PROGRAM Stn3
VAR

	start3: BOOL;
	reset3: BOOL;

	Stn3ProcessFE: F_TRIG;
	Stn3ProcessRE: R_TRIG;
	bCutStn3ProcessHalt: BOOL;
	DoorClose3: R_TRIG;
	bStn3DoorClamp: BOOL;
END_VAR
VAR // added by the converter: edge detectors and wires of the graphical bodies
    _w1, _w2 : ANY;
    _w3 : BOOL;
END_VAR

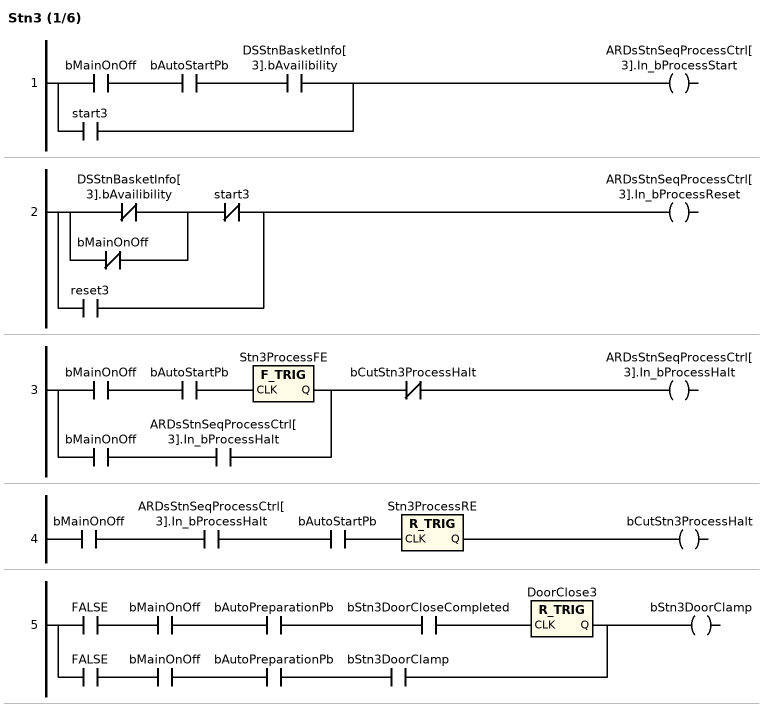
// NETWORK 1
ARDsStnSeqProcessCtrl[3].In_bProcessStart := bMainOnOff AND bAutoStartPb AND DSStnBasketInfo[3].bAvailibility OR start3;

// NETWORK 2
ARDsStnSeqProcessCtrl[3].In_bProcessReset := (NOT DSStnBasketInfo[3].bAvailibility OR NOT bMainOnOff) AND NOT start3 OR reset3;

// NETWORK 3
Stn3ProcessFE(CLK := bMainOnOff AND bAutoStartPb); // F_TRIG
ARDsStnSeqProcessCtrl[3].In_bProcessHalt := (Stn3ProcessFE.Q OR bMainOnOff AND ARDsStnSeqProcessCtrl[3].In_bProcessHalt) AND NOT bCutStn3ProcessHalt;

// NETWORK 4
Stn3ProcessRE(CLK := bMainOnOff AND ARDsStnSeqProcessCtrl[3].In_bProcessHalt AND bAutoStartPb); // R_TRIG
bCutStn3ProcessHalt := Stn3ProcessRE.Q;

// NETWORK 5
DoorClose3(CLK := (FALSE AND bMainOnOff AND bAutoPreparationPb) AND bStn3DoorCloseCompleted); // R_TRIG
bStn3DoorClamp := DoorClose3.Q OR (FALSE AND bMainOnOff AND bAutoPreparationPb) AND bStn3DoorClamp;

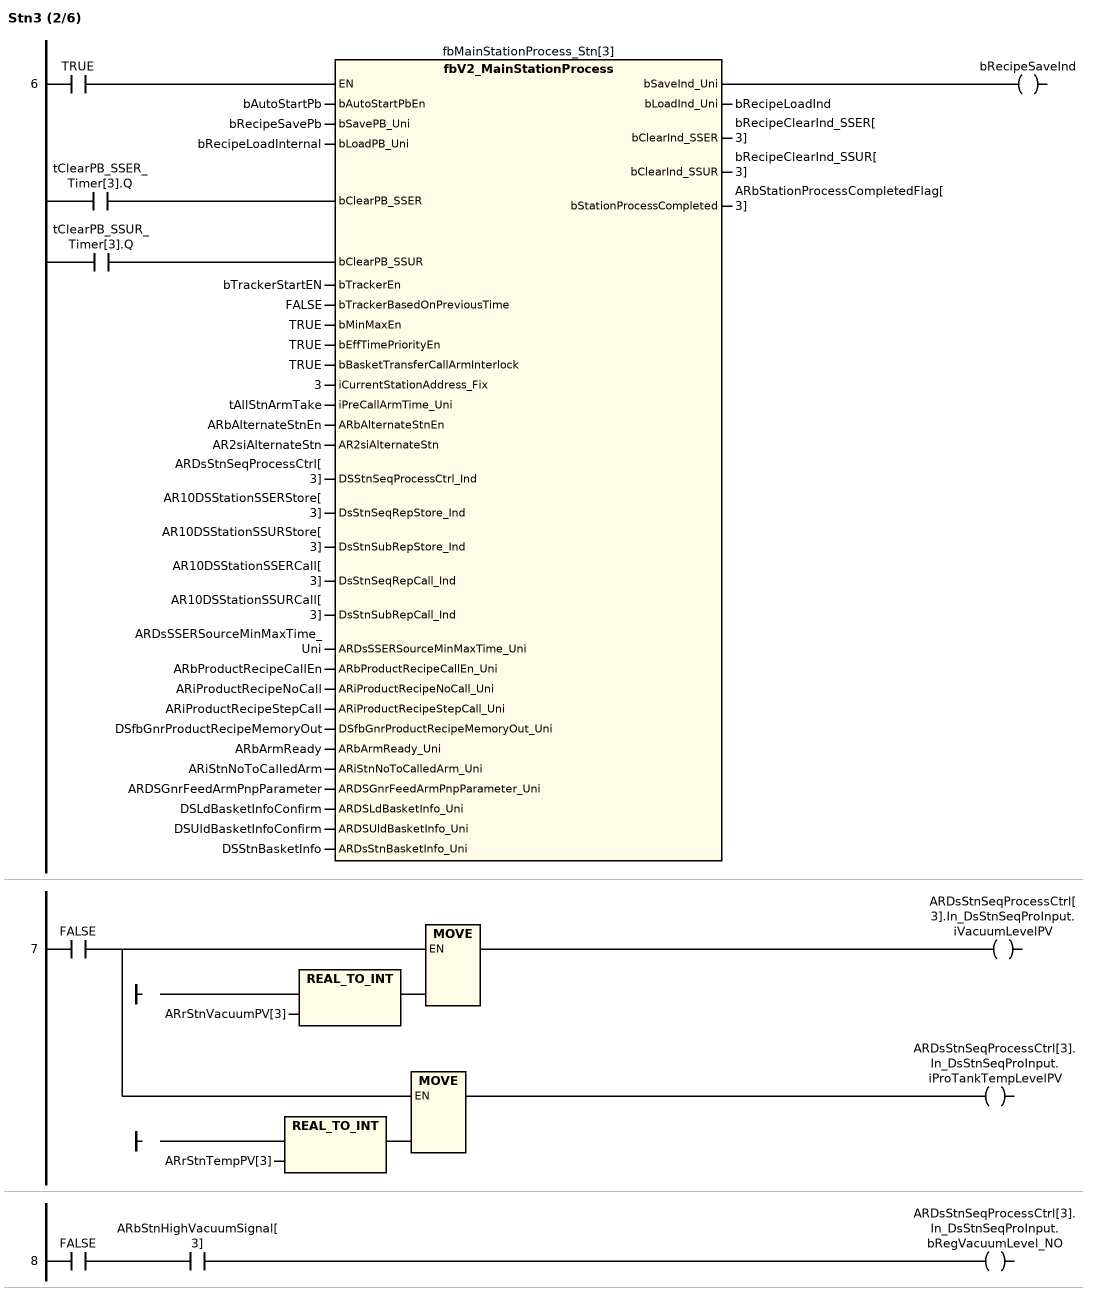
// NETWORK 6
fbMainStationProcess_Stn[3](
    bAutoStartPbEn := bAutoStartPb,
    bSavePB_Uni := bRecipeSavePb,
    bLoadPB_Uni := bRecipeLoadInternal,
    bClearPB_SSER := tClearPB_SSER_Timer[3].Q,
    bClearPB_SSUR := tClearPB_SSUR_Timer[3].Q,
    bTrackerEn := bTrackerStartEN,
    bTrackerBasedOnPreviousTime := FALSE,
    bMinMaxEn := TRUE,
    bEffTimePriorityEn := TRUE,
    bBasketTransferCallArmInterlock := TRUE,
    iCurrentStationAddress_Fix := 3,
    iPreCallArmTime_Uni := tAllStnArmTake,
    ARbAlternateStnEn := ARbAlternateStnEn,
    AR2siAlternateStn := AR2siAlternateStn,
    DSStnSeqProcessCtrl_Ind := ARDsStnSeqProcessCtrl[3],
    DsStnSeqRepStore_Ind := AR10DSStationSSERStore[3],
    DsStnSubRepStore_Ind := AR10DSStationSSURStore[3],
    DsStnSeqRepCall_Ind := AR10DSStationSSERCall[3],
    DsStnSubRepCall_Ind := AR10DSStationSSURCall[3],
    ARDsSSERSourceMinMaxTime_Uni := ARDsSSERSourceMinMaxTime_Uni,
    ARbProductRecipeCallEn_Uni := ARbProductRecipeCallEn,
    ARiProductRecipeNoCall_Uni := ARiProductRecipeNoCall,
    ARiProductRecipeStepCall_Uni := ARiProductRecipeStepCall,
    DSfbGnrProductRecipeMemoryOut_Uni := DSfbGnrProductRecipeMemoryOut,
    ARbArmReady_Uni := ARbArmReady,
    ARiStnNoToCalledArm_Uni := ARiStnNoToCalledArm,
    ARDSGnrFeedArmPnpParameter_Uni := ARDSGnrFeedArmPnpParameter,
    ARDSLdBasketInfo_Uni := DSLdBasketInfoConfirm,
    ARDSUldBasketInfo_Uni := DSUldBasketInfoConfirm,
    ARDsStnBasketInfo_Uni := DSStnBasketInfo,
    bLoadInd_Uni => bRecipeLoadInd,
    bClearInd_SSER => bRecipeClearInd_SSER[3],
    bClearInd_SSUR => bRecipeClearInd_SSUR[3],
    bStationProcessCompleted => ARbStationProcessCompletedFlag[3]); // fbV2_MainStationProcess
bRecipeSaveInd := fbMainStationProcess_Stn[3].bSaveInd_Uni;

// NETWORK 7
IF FALSE THEN _w1 := REAL_TO_INT(ARrStnVacuumPV[3]); END_IF
ARDsStnSeqProcessCtrl[3].In_DsStnSeqProInput.iVacuumLevelPV := _w1;
IF FALSE THEN _w2 := REAL_TO_INT(ARrStnTempPV[3]); END_IF
ARDsStnSeqProcessCtrl[3].In_DsStnSeqProInput.iProTankTempLevelPV := _w2;

// NETWORK 8
ARDsStnSeqProcessCtrl[3].In_DsStnSeqProInput.bRegVacuumLevel_NO := FALSE AND ARbStnHighVacuumSignal[3];

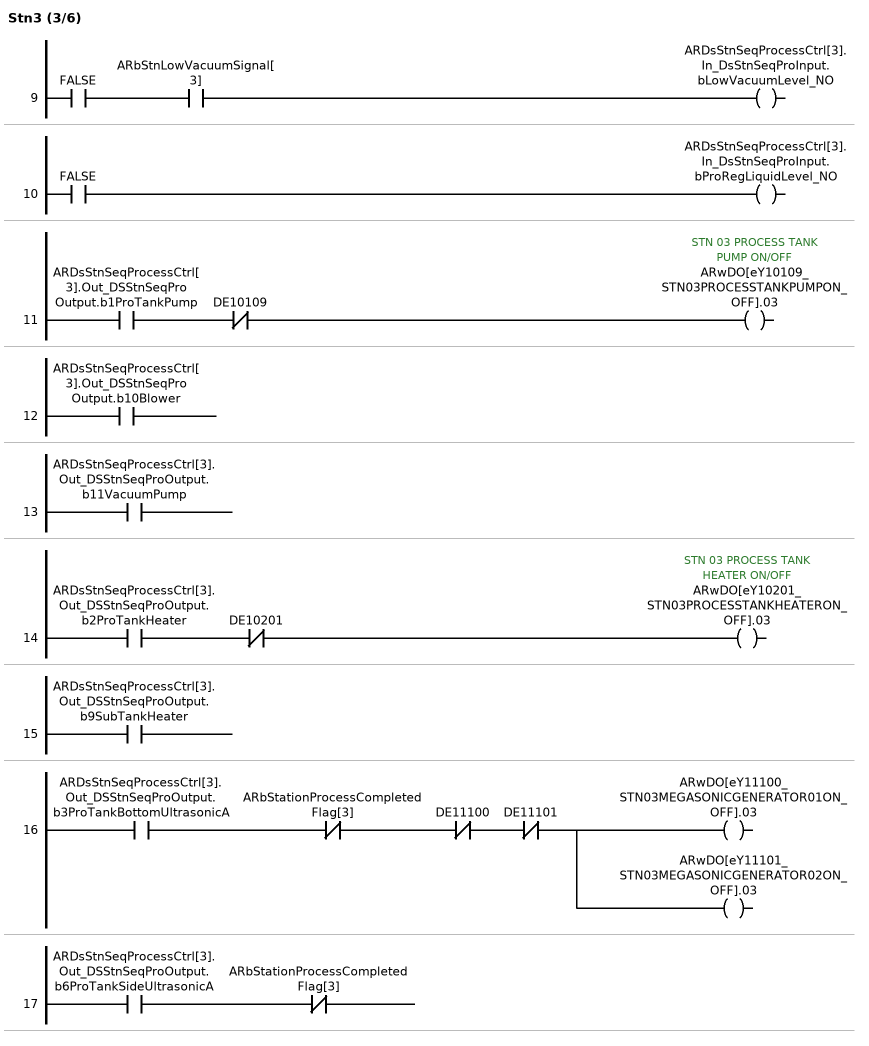
// NETWORK 9
ARDsStnSeqProcessCtrl[3].In_DsStnSeqProInput.bLowVacuumLevel_NO := FALSE AND ARbStnLowVacuumSignal[3];

// NETWORK 10
ARDsStnSeqProcessCtrl[3].In_DsStnSeqProInput.bProRegLiquidLevel_NO := FALSE;

// NETWORK 11
//   ARwDO[eY10109_STN03PROCESSTANKPUMPON_OFF].03: STN 03 PROCESS TANK PUMP ON/OFF
ARwDO[eY10109_STN03PROCESSTANKPUMPON_OFF].03 := ARDsStnSeqProcessCtrl[3].Out_DSStnSeqProOutput.b1ProTankPump AND NOT DE10109;

// NETWORK 12
(* ARDsStnSeqProcessCtrl[3].Out_DSStnSeqProOutput.b10Blower; not connected *)

// NETWORK 13
(* ARDsStnSeqProcessCtrl[3].Out_DSStnSeqProOutput.b11VacuumPump; not connected *)

// NETWORK 14
//   ARwDO[eY10201_STN03PROCESSTANKHEATERON_OFF].03: STN 03 PROCESS TANK HEATER ON/OFF
ARwDO[eY10201_STN03PROCESSTANKHEATERON_OFF].03 := ARDsStnSeqProcessCtrl[3].Out_DSStnSeqProOutput.b2ProTankHeater AND NOT DE10201;

// NETWORK 15
(* ARDsStnSeqProcessCtrl[3].Out_DSStnSeqProOutput.b9SubTankHeater; not connected *)

// NETWORK 16
_w3 := ARDsStnSeqProcessCtrl[3].Out_DSStnSeqProOutput.b3ProTankBottomUltrasonicA AND NOT ARbStationProcessCompletedFlag[3] AND NOT DE11100 AND NOT DE11101;
ARwDO[eY11100_STN03MEGASONICGENERATOR01ON_OFF].03 := _w3;
ARwDO[eY11101_STN03MEGASONICGENERATOR02ON_OFF].03 := _w3;

// NETWORK 17
(* ARDsStnSeqProcessCtrl[3].Out_DSStnSeqProOutput.b6ProTankSideUltrasonicA AND NOT ARbStationProcessCompletedFlag[3]; result not used *)

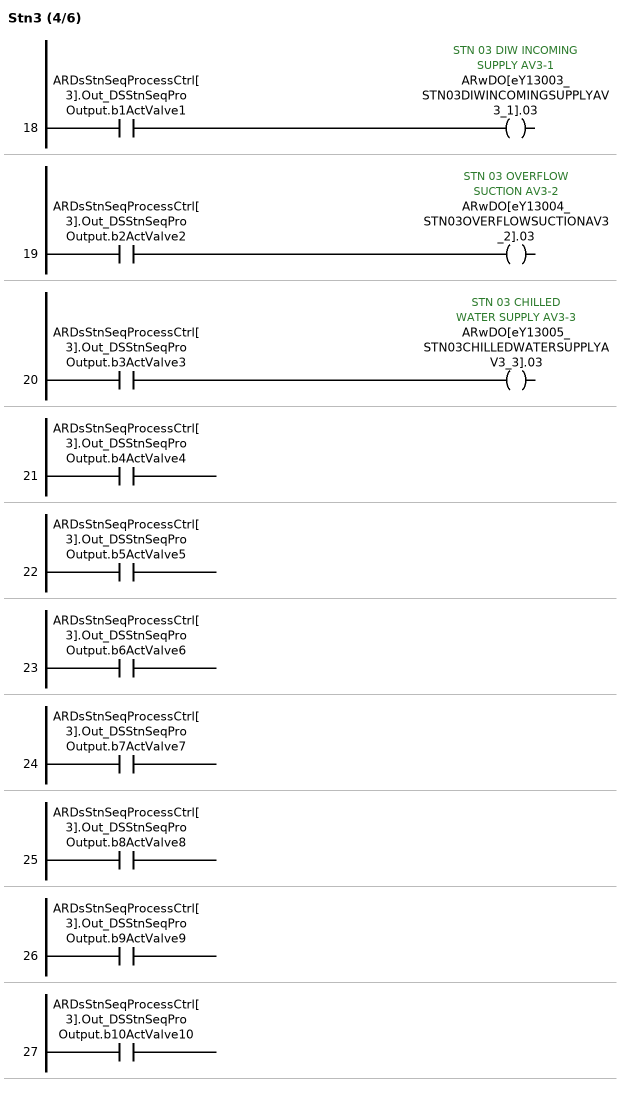
// NETWORK 18
//   ARwDO[eY13003_STN03DIWINCOMINGSUPPLYAV3_1].03: STN 03 DIW INCOMING SUPPLY AV3-1
ARwDO[eY13003_STN03DIWINCOMINGSUPPLYAV3_1].03 := ARDsStnSeqProcessCtrl[3].Out_DSStnSeqProOutput.b1ActValve1;

// NETWORK 19
//   ARwDO[eY13004_STN03OVERFLOWSUCTIONAV3_2].03: STN 03 OVERFLOW SUCTION AV3-2
ARwDO[eY13004_STN03OVERFLOWSUCTIONAV3_2].03 := ARDsStnSeqProcessCtrl[3].Out_DSStnSeqProOutput.b2ActValve2;

// NETWORK 20
//   ARwDO[eY13005_STN03CHILLEDWATERSUPPLYAV3_3].03: STN 03 CHILLED WATER SUPPLY AV3-3
ARwDO[eY13005_STN03CHILLEDWATERSUPPLYAV3_3].03 := ARDsStnSeqProcessCtrl[3].Out_DSStnSeqProOutput.b3ActValve3;

// NETWORK 21
(* ARDsStnSeqProcessCtrl[3].Out_DSStnSeqProOutput.b4ActValve4; not connected *)

// NETWORK 22
(* ARDsStnSeqProcessCtrl[3].Out_DSStnSeqProOutput.b5ActValve5; not connected *)

// NETWORK 23
(* ARDsStnSeqProcessCtrl[3].Out_DSStnSeqProOutput.b6ActValve6; not connected *)

// NETWORK 24
(* ARDsStnSeqProcessCtrl[3].Out_DSStnSeqProOutput.b7ActValve7; not connected *)

// NETWORK 25
(* ARDsStnSeqProcessCtrl[3].Out_DSStnSeqProOutput.b8ActValve8; not connected *)

// NETWORK 26
(* ARDsStnSeqProcessCtrl[3].Out_DSStnSeqProOutput.b9ActValve9; not connected *)

// NETWORK 27
(* ARDsStnSeqProcessCtrl[3].Out_DSStnSeqProOutput.b10ActValve10; not connected *)

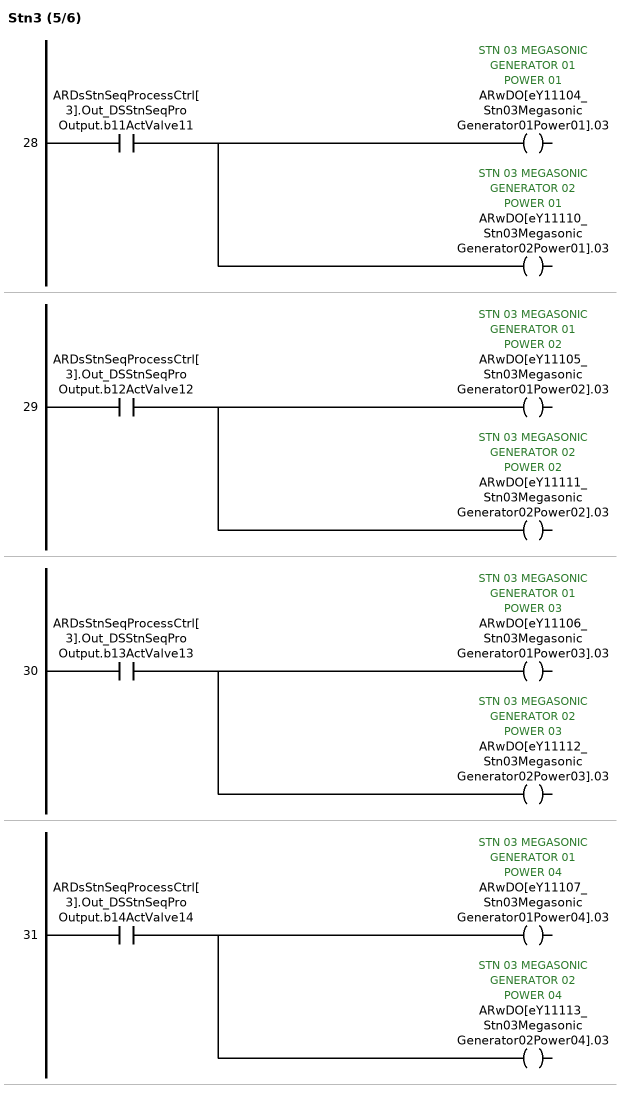
// NETWORK 28
//   ARwDO[eY11104_Stn03MegasonicGenerator01Power01].03: STN 03 MEGASONIC GENERATOR 01 POWER 01
//   ARwDO[eY11110_Stn03MegasonicGenerator02Power01].03: STN 03 MEGASONIC GENERATOR 02 POWER 01
ARwDO[eY11104_Stn03MegasonicGenerator01Power01].03 := ARDsStnSeqProcessCtrl[3].Out_DSStnSeqProOutput.b11ActValve11;
ARwDO[eY11110_Stn03MegasonicGenerator02Power01].03 := ARDsStnSeqProcessCtrl[3].Out_DSStnSeqProOutput.b11ActValve11;

// NETWORK 29
//   ARwDO[eY11105_Stn03MegasonicGenerator01Power02].03: STN 03 MEGASONIC GENERATOR 01 POWER 02
//   ARwDO[eY11111_Stn03MegasonicGenerator02Power02].03: STN 03 MEGASONIC GENERATOR 02 POWER 02
ARwDO[eY11105_Stn03MegasonicGenerator01Power02].03 := ARDsStnSeqProcessCtrl[3].Out_DSStnSeqProOutput.b12ActValve12;
ARwDO[eY11111_Stn03MegasonicGenerator02Power02].03 := ARDsStnSeqProcessCtrl[3].Out_DSStnSeqProOutput.b12ActValve12;

// NETWORK 30
//   ARwDO[eY11106_Stn03MegasonicGenerator01Power03].03: STN 03 MEGASONIC GENERATOR 01 POWER 03
//   ARwDO[eY11112_Stn03MegasonicGenerator02Power03].03: STN 03 MEGASONIC GENERATOR 02 POWER 03
ARwDO[eY11106_Stn03MegasonicGenerator01Power03].03 := ARDsStnSeqProcessCtrl[3].Out_DSStnSeqProOutput.b13ActValve13;
ARwDO[eY11112_Stn03MegasonicGenerator02Power03].03 := ARDsStnSeqProcessCtrl[3].Out_DSStnSeqProOutput.b13ActValve13;

// NETWORK 31
//   ARwDO[eY11107_Stn03MegasonicGenerator01Power04].03: STN 03 MEGASONIC GENERATOR 01 POWER 04
//   ARwDO[eY11113_Stn03MegasonicGenerator02Power04].03: STN 03 MEGASONIC GENERATOR 02 POWER 04
ARwDO[eY11107_Stn03MegasonicGenerator01Power04].03 := ARDsStnSeqProcessCtrl[3].Out_DSStnSeqProOutput.b14ActValve14;
ARwDO[eY11113_Stn03MegasonicGenerator02Power04].03 := ARDsStnSeqProcessCtrl[3].Out_DSStnSeqProOutput.b14ActValve14;

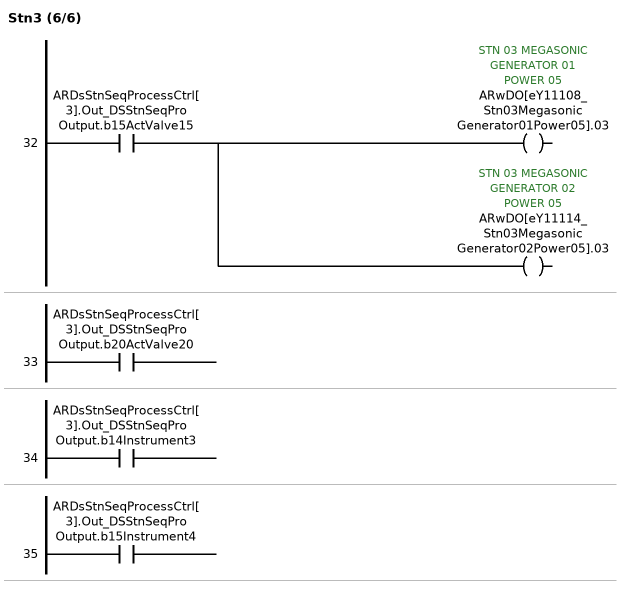
// NETWORK 32
//   ARwDO[eY11108_Stn03MegasonicGenerator01Power05].03: STN 03 MEGASONIC GENERATOR 01 POWER 05
//   ARwDO[eY11114_Stn03MegasonicGenerator02Power05].03: STN 03 MEGASONIC GENERATOR 02 POWER 05
ARwDO[eY11108_Stn03MegasonicGenerator01Power05].03 := ARDsStnSeqProcessCtrl[3].Out_DSStnSeqProOutput.b15ActValve15;
ARwDO[eY11114_Stn03MegasonicGenerator02Power05].03 := ARDsStnSeqProcessCtrl[3].Out_DSStnSeqProOutput.b15ActValve15;

// NETWORK 33
(* ARDsStnSeqProcessCtrl[3].Out_DSStnSeqProOutput.b20ActValve20; not connected *)

// NETWORK 34
(* ARDsStnSeqProcessCtrl[3].Out_DSStnSeqProOutput.b14Instrument3; not connected *)

// NETWORK 35
(* ARDsStnSeqProcessCtrl[3].Out_DSStnSeqProOutput.b15Instrument4; not connected *)

END_PROGRAM

(* stored: Version 1.1.0.1, ProductVersion 3.1.4024.12
   POU Stn3: Id {79d5c1cb-0b47-401d-85fd-2150156bffcd}, SpecialFunc None *)
